TYPE ST_P_COMPLETE_OP :
STRUCT
	SetIndex:				BOOL;
	Index:					INT;
	Barcode:			INT;
END_STRUCT
END_TYPE

(* stored: Version 1.1.0.1, ProductVersion 3.1.4024.10
   DUT ST_P_COMPLETE_OP: Id {ee2ba148-cc59-460e-b1ee-1d81002d13f0} *)
